FUNCTION RawToVoltage : REAL
VAR_INPUT
	raw : UINT;            // 0..6000
END_VAR


RawToVoltage := UINT_TO_REAL(raw) * 0.01;  // → 0.00…60.00 V

END_FUNCTION

(* stored: Version 1.1.0.1
   POU RawToVoltage: Id {576a5706-8be0-43f1-83e2-dc930bc13e71}, SpecialFunc None *)
